{attribute 'linkalways'} 
{attribute 'no_explicit_call' := 'This FB is a CLASS and must be accessed using methods or properties'}
{attribute 'enable_dynamic_creation'}
FUNCTION_BLOCK FINAL NE_WORD EXTENDS Node
VAR
	in1 : _WORD(0);
	in2 : _WORD(0);
	out : _BOOL(FALSE);
END_VAR

METHOD PUBLIC Clone : I_Node
VAR
	pNode : POINTER TO NE_WORD;
END_VAR
pNode := __NEW(NE_WORD);
Clone := pNode^;
END_METHOD

METHOD FB_init : BOOL
VAR_INPUT
	bInitRetains : BOOL; // if TRUE, the retain variables are initialized (warm start / cold start)
	bInCopyCode : BOOL;  // if TRUE, the instance afterwards gets moved into the copy code (online change)
END_VAR
AddInput('in1',THIS^.in1);
AddInput('in2',THIS^.in2);
AddOutput('out', THIS^.out);
END_METHOD

METHOD PROTECTED OnExecute
VAR
END_VAR
out.Value := in1.Value <> in2.Value;
END_METHOD

END_FUNCTION_BLOCK

(* stored: Version 1.1.0.1, ProductVersion 3.1.4024.15
   POU NE_WORD: Id {715aeb63-d113-4f20-8590-9a233d61fdb8}, SpecialFunc None
   Folder Constructor: Id {c67092ab-22e7-4523-8294-4e28a7efda8e}
   Method Clone: Id {aaca0101-2d07-4f77-8478-0444f6aaabce}
   Method FB_init: Id {ff033d24-c91a-42a1-a6c0-94bd8bf5adc4}
   Method OnExecute: Id {45cc30a7-15a3-4a06-a621-a49fe35360bc} *)
